# B&R Automation Studio project mappCleanUp
Automation Studio 4.10.6.39 SP

## Configuration Config1

CPU PC_any, AutomationRuntime B4.91, Build 4.1.2, Vc V4.73.0

### Task classes (Cpu.sw)
```
Cyclic#8 (cycle 10000 us):
  mappCleanU <- mappCleanUp.prg
Binaries: FWRules, TCData, udbdef, asfw, User, iomap, sysconf, arconfig, ashwd, Role, ashwac
Libraries: sys_lib, runtime, FileIO, AsBrStr, IecCheck, standard, asieccon, astime
```

### Hardware
```
PC : PC_any v1.1.1.0 (OrderNumber=PC)
  ConfigurationID = mappCleanUp_Config1
  Cyclic8Duration = 10000
  FileDevice1
  FileDeviceName1 = USER_PATH
  FileDevicePath1 = c:\Temp\CleanUpTest
```

## Configuration Simulation

CPU PC_any, AutomationRuntime M4.93, Build 4.1.2, Vc V4.73.0

### Hardware
```
PC : PC_any v1.1.1.0 (OrderNumber=PC)
  ConfigurationID = mappCleanUp_Config1
  Cyclic8Duration = 10000
  FileDevice1
  FileDeviceName1 = USER
  FileDevicePath1 = c:\Temp\CleanUpTest
```

## Configuration X20CP

CPU X20CP3687X, AutomationRuntime M4.93, Build 4.1.2, Vc V4.73.3

### Task classes (Cpu.sw)
```
Cyclic#8:
  mappCleanU <- mappCleanUp.prg
Libraries: operator, runtime, astime, AsIecCon, sys_lib, FileIO, AsBrStr, IecCheck, standard
```

### Hardware
```
X20CP3687X : X20CP3687X v1.8.2.0
  Connector IF2:
    ActivateDevice = 1
    ActivateSnmp = 2
  ConfigurationID = mappCleanUp_X20CP
  FileDevice1
  FileDeviceName1 = USER
  FileDevicePath1 = USER_PATH
  FtpUser1
  FtpUsername1 = admin
  FtpUserPassword1 = +ZKvy1J8o41WeGJ4ICTiSOGGvLAHu+nBthxiKzD2AAg=  // admin
  FtpUserSalt1 = TuKBiUW7
  FTPAccessRight1 = 0
```

## Logical view

Binary libraries used (declarations not repeated): operator, runtime, astime, AsIecCon, sys_lib, FileIO, AsBrStr, IecCheck, standard


### Program Logical/mappCleanUp (IEC)

#### Main.st - Init, cyclic, exit code
```iecst
PROGRAM _INIT
	(* Insert code here *)

END_PROGRAM

PROGRAM _CYCLIC
	CASE State OF
		CLEANUP_WAIT:
			CleanUp.Status := ERR_OK;

			DevMemInfo_0.enable := FALSE;
			DevMemInfo_0();
			DirInfo_0.enable := FALSE;
			DirInfo_0();
			DirOpen_0.enable := FALSE;
			DirOpen_0();
			DirReadEx_0.enable := FALSE;
			DirReadEx_0();
			DirClose_0.enable := FALSE;
			DirClose_0();
			FileDelete_0.enable := FALSE;
			FileDelete_0();

			// Command delete oldest file
			IF EDGEPOS(CleanUp.CMD.DeleteOldest) THEN
				// Reset variables
				brsmemset(ADR(CleanUp.DAT), 0, SIZEOF(CleanUp.DAT));
				brsmemset(ADR(FileInformation), 0, SIZEOF(FileInformation));

				// Set callbacks and status
				StateAfterInfo := CLEANUP_DIR_INFO;
				StateAfterRead := CLEANUP_DELETE_OLDEST;
				StateAfterDelete := CLEANUP_DIR_CLOSE;
				CleanUp.Status := ERR_FUB_BUSY;

				State := CLEANUP_MEM_INFO;
			END_IF

			// Command delete oldest than
			IF EDGEPOS(CleanUp.CMD.DeleteOlderThan) THEN
				IF CleanUp.PAR.OlderThan <> DT#1970-01-01-00:00:00 THEN
					// Reset variables
					brsmemset(ADR(CleanUp.DAT), 0, SIZEOF(CleanUp.DAT));
					brsmemset(ADR(FileInformation), 0, SIZEOF(FileInformation));

					// Set callbacks and status
					StateAfterInfo := CLEANUP_DIR_INFO;
					StateAfterRead := CLEANUP_DELETE_OLDER_THAN;
					StateAfterDelete := CLEANUP_DIR_READ;
					CleanUp.Status := ERR_FUB_BUSY;

					State := CLEANUP_MEM_INFO;
				ELSE
					State := CreateError(ADR(CleanUp), CLEANUP_ERR_PAR_IS_EMPTY, 'parameter >OlderThan< was not set', State, ADR(Logger));
				END_IF
			END_IF

			// Command delete files and keep x
			IF EDGEPOS(CleanUp.CMD.DeleteMaxFiles) THEN
				IF CleanUp.PAR.MaxFilesToKeep <> 0 THEN
					// Reset variables
					brsmemset(ADR(CleanUp.DAT), 0, SIZEOF(CleanUp.DAT));
					brsmemset(ADR(FileInformation), 0, SIZEOF(FileInformation));
					SimFileCount := 0;

					// Set callbacks and status
					StateAfterInfo := CLEANUP_DIR_INFO;
					StateAfterRead := CLEANUP_DELETE_MAX_FILES_1;
					StateAfterDelete := CLEANUP_DELETE_MAX_FILES_2;

					CleanUp.Status := ERR_FUB_BUSY;

					State := CLEANUP_MEM_INFO;
				ELSE
					State := CreateError(ADR(CleanUp), CLEANUP_ERR_PAR_IS_EMPTY, 'parameter >MaxFilesToKeep< was not set', State, ADR(Logger));
				END_IF
			END_IF

			// Command delete files until minimum memory is restored
			IF EDGEPOS(CleanUp.CMD.DeleteMinSpace) THEN
				IF CleanUp.PAR.MinSpace <> 0 THEN
					// Reset variables
					brsmemset(ADR(CleanUp.DAT), 0, SIZEOF(CleanUp.DAT));
					brsmemset(ADR(FileInformation), 0, SIZEOF(FileInformation));
					SimMemCount := 0;

					// Set callbacks and status
					StateAfterInfo := CLEANUP_DIR_INFO;
					StateAfterRead := CLEANUP_DELETE_MIN_SPACE_1;
					StateAfterDelete := CLEANUP_DELETE_MIN_SPACE_2;

					CleanUp.Status := ERR_FUB_BUSY;

					State := CLEANUP_MEM_INFO;
				ELSE
					State := CreateError(ADR(CleanUp), CLEANUP_ERR_PAR_IS_EMPTY, 'parameter >MinSpace< was not set', State, ADR(Logger));
				END_IF
			END_IF

			// Command update free space
			IF EDGEPOS(CleanUp.CMD.UpdateFreeSpace) THEN
				// Set callbacks
				StateAfterInfo := CLEANUP_WAIT;

				State := CLEANUP_MEM_INFO;
			END_IF

			// -------------------------------------------------------------------------------------------
			// Get device information
		CLEANUP_MEM_INFO:
			DevMemInfo_0.enable := TRUE;
			DevMemInfo_0.pDevice := ADR(CleanUp.PAR.Device);
			DevMemInfo_0();

			// Memory information successful
			IF DevMemInfo_0.status = ERR_OK THEN
				CleanUp.DAT.FreeSpace := DevMemInfo_0.freemem + (SimMemCount * CleanUp.PAR.Simulate);

				// Go to next step
				State := StateAfterInfo;

			// Error
			ELSIF DevMemInfo_0.status <> ERR_FUB_BUSY THEN
				TmpStr1 := 'ERR memory info > ';
				brsstrcat(ADR(TmpStr1), ADR(CleanUp.PAR.Device));
				State := CreateError(ADR(CleanUp), DevMemInfo_0.status, TmpStr1, State, ADR(Logger));
			END_IF

			// -------------------------------------------------------------------------------------------
			// Get folder information
		CLEANUP_DIR_INFO:
			DirInfo_0.enable := TRUE;
			DirInfo_0.pDevice := ADR(CleanUp.PAR.Device);
			DirInfo_0.pPath := ADR(CleanUp.PAR.Path);
			DirInfo_0();

			// Dir info successful
			IF DirInfo_0.status = ERR_OK THEN
				CleanUp.DAT.FilesCount := DirInfo_0.filenum;

				// Go to next step
				State := CLEANUP_DIR_OPEN;

			// Error
			ELSIF DirInfo_0.status <> ERR_FUB_BUSY THEN
				TmpStr1 := 'ERR dir info > ';
				brsstrcat(ADR(TmpStr1), ADR(CleanUp.PAR.Device));
				brsstrcat(ADR(TmpStr1), ADR(' with dir > '));
				brsstrcat(ADR(TmpStr1), ADR(CleanUp.PAR.Path));
				State := CreateError(ADR(CleanUp), DirInfo_0.status, TmpStr1, State, ADR(Logger));
			END_IF

			// -------------------------------------------------------------------------------------------
			// Start reading folder
		CLEANUP_DIR_OPEN:
			DirOpen_0.enable := TRUE;
			DirOpen_0.pDevice := ADR(CleanUp.PAR.Device);
			DirOpen_0.pName := ADR(CleanUp.PAR.Path);
			DirOpen_0();

			// Dir open successful
			IF DirOpen_0.status = ERR_OK THEN
				// Generate log entry
				TmpStr1 := 'open device > ';
				brsstrcat(ADR(TmpStr1), ADR(CleanUp.PAR.Device));
				brsstrcat(ADR(TmpStr1), ADR(' with dir > '));
				brsstrcat(ADR(TmpStr1), ADR(CleanUp.PAR.Path));
				CreateLoggerEntry(ADR(TmpStr1), ADR(Logger));

				// Go to next step
				State := CLEANUP_DIR_READ;

				// Error
			ELSIF DirOpen_0.status <> ERR_FUB_BUSY THEN
				TmpStr1 := 'ERR open device > ';
				brsstrcat(ADR(TmpStr1), ADR(CleanUp.PAR.Device));
				brsstrcat(ADR(TmpStr1), ADR(' with dir > '));
				brsstrcat(ADR(TmpStr1), ADR(CleanUp.PAR.Path));
				State := CreateError(ADR(CleanUp), DirOpen_0.status, TmpStr1, State, ADR(Logger));
			END_IF

			// -------------------------------------------------------------------------------------------
			// Start reading folder
		CLEANUP_DIR_READ:
			DirReadEx_0.enable := TRUE;
			DirReadEx_0.ident := DirOpen_0.ident;
			DirReadEx_0.pData := ADR(FileDirInfo);
			DirReadEx_0.data_len := SIZEOF(FileDirInfo);
			DirReadEx_0();

			// New file found
			IF DirReadEx_0.status = ERR_OK AND FileDirInfo.Mode = fiFILE THEN
				IF brsstrcmp(ADR(FileDirInfo.Filename), ADR('.')) <> 0 AND brsstrcmp(ADR(FileDirInfo.Filename), ADR('..')) <> 0 THEN

					// Check if file name matches pattern
					IF IsInstr(ADR(FileDirInfo.Filename), ADR(CleanUp.PAR.Pattern)) OR CleanUp.PAR.Pattern = '' THEN
						// Generate log entry
						TmpStr1 := 'found file > ';
						brsstrcat(ADR(TmpStr1), ADR(FileDirInfo.Filename));
						CreateLoggerEntry(ADR(TmpStr1), ADR(Logger));

						// Go to next state
						State := StateAfterRead;
					ELSE
						// Generate log entry
						TmpStr1 := 'file does not match pattern > ';
						brsstrcat(ADR(TmpStr1), ADR(FileDirInfo.Filename));
						CreateLoggerEntry(ADR(TmpStr1), ADR(Logger));
					END_IF

					DirReadEx_0.enable := FALSE;
					DirReadEx_0();

				END_IF

			// No more entries
			ELSIF DirReadEx_0.status = fiERR_NO_MORE_ENTRIES THEN
				// Generate log entry
				CreateLoggerEntry(ADR('no more files found '), ADR(Logger));

				// Go to next state
				State := StateAfterRead;

				// Error
			ELSIF DirReadEx_0.status <> ERR_OK AND DirReadEx_0.status <> ERR_FUB_BUSY THEN
				TmpStr1 := 'ERR open file > ';
				brsstrcat(ADR(TmpStr1), ADR(FileDirInfo.Filename));
				State := CreateError(ADR(CleanUp), DirReadEx_0.status, TmpStr1, State, ADR(Logger));
			END_IF

			// -------------------------------------------------------------------------------------------
			// Delete oldest file
		CLEANUP_DELETE_OLDEST:
			// Evaluate next file
			IF DirReadEx_0.status <> fiERR_NO_MORE_ENTRIES THEN
				// File must be older than last
				IF FileInformation.Date > FileDirInfo.Date OR FileInformation.Date = DT#1970-01-01-00:00:00 THEN
					// Pretend that files were delete in simulation mode
					IF CleanUp.PAR.Simulate AND i < SIZEOF(CleanUp.DAT.FilesList)/SIZEOF(CleanUp.DAT.FilesList[0]) THEN
						i := 0;
						WHILE i <= CleanUp.DAT.FilesDeleted DO
							IF brsstrcmp(ADR(CleanUp.DAT.FilesList[i]), ADR(FileDirInfo.Filename)) = 0 THEN
								EXIT;
							END_IF
							i := i + 1;
						END_WHILE;
					ELSE
						i := CleanUp.DAT.FilesDeleted + 1;
					END_IF
					IF i = CleanUp.DAT.FilesDeleted + 1 THEN
						FileInformation := FileDirInfo;
					END_IF
				END_IF
				State := CLEANUP_DIR_READ;

			// Delete oldest file
			ELSE
				// Make sure we found at least one entry
				IF FileInformation.Date <> DT#1970-01-01-00:00:00 THEN
					// Fake simulation values
					IF CleanUp.PAR.Simulate THEN
						SimFileCount := SimFileCount + 1;
						SimMemCount := SimMemCount + FileInformation.Filelength;
					END_IF
					brsstrcpy(ADR(FileDeleteName), ADR(FileInformation.Filename));
					State := CLEANUP_FILE_DELETE;
				ELSE
					// Create error when there are not enough files to delete
					IF CleanUp.CMD.DeleteMinSpace AND DevMemInfo_0.freemem + SimMemCount < CleanUp.PAR.MinSpace THEN
						State := CreateError(ADR(CleanUp), CLEANUP_ERR_MIN_SPACE, 'Minimum space could not be achieved', State, ADR(Logger));
					ELSIF CleanUp.CMD.DeleteMaxFiles AND DirInfo_0.filenum - SimFileCount > CleanUp.PAR.MaxFilesToKeep THEN
						State := CreateError(ADR(CleanUp), CLEANUP_ERR_MIN_FILES, 'Minimum file count could not be achieved', State, ADR(Logger));
					ELSE
						State := CLEANUP_DIR_CLOSE;
					END_IF
				END_IF
			END_IF

			// -------------------------------------------------------------------------------------------
			// Delete files older than x
		CLEANUP_DELETE_OLDER_THAN:
			// Read next file, remember oldest file
			IF DirReadEx_0.status <> fiERR_NO_MORE_ENTRIES THEN
				IF FileDirInfo.Date > CleanUp.PAR.OlderThan THEN
					brsstrcpy(ADR(FileDeleteName), ADR(FileDirInfo.Filename));
					FileInformation := FileDirInfo;
					State := CLEANUP_FILE_DELETE;
				ELSE
					State := CLEANUP_DIR_READ;
				END_IF

				// Finish deleting old files
			ELSE
				State := CLEANUP_DIR_CLOSE;
			END_IF

			// -------------------------------------------------------------------------------------------
			// Delete files and keep x
		CLEANUP_DELETE_MAX_FILES_1:
			// Read next file, remember oldest file
			IF DirInfo_0.filenum - SimFileCount > CleanUp.PAR.MaxFilesToKeep THEN
				StateAfterRead := CLEANUP_DELETE_OLDEST;
				State := CLEANUP_DELETE_OLDEST;

			// Finish deleting old files
			ELSE
				State := CLEANUP_DIR_CLOSE;
			END_IF

			// -------------------------------------------------------------------------------------------
			// Delete files and keep x
		CLEANUP_DELETE_MAX_FILES_2:
			brsmemset(ADR(FileInformation), 0, SIZEOF(FileInformation));
			DirInfo_0.enable := FALSE;
			DirInfo_0();

			StateAfterRead := CLEANUP_DELETE_MAX_FILES_1;
			State := CLEANUP_DIR_INFO;

			// -------------------------------------------------------------------------------------------
			// Delete files until minimum free space is restored
		CLEANUP_DELETE_MIN_SPACE_1:
			// Read next file, remember oldest file
			IF DevMemInfo_0.freemem + SimMemCount < CleanUp.PAR.MinSpace THEN
				StateAfterRead := CLEANUP_DELETE_OLDEST;
				State := CLEANUP_DELETE_OLDEST;

			// Finish deleting old files
			ELSE
				State := CLEANUP_DIR_CLOSE;
			END_IF

			// -------------------------------------------------------------------------------------------
			// Delete files until minimum free space is restored
		CLEANUP_DELETE_MIN_SPACE_2:
			brsmemset(ADR(FileInformation), 0, SIZEOF(FileInformation));
			DirInfo_0.enable := FALSE;
			DirInfo_0();

			StateAfterRead := CLEANUP_DELETE_MIN_SPACE_1;
			State := CLEANUP_MEM_INFO;

			// -------------------------------------------------------------------------------------------
			// Close dir read
		CLEANUP_DIR_CLOSE:
			DirClose_0.enable := TRUE;
			DirClose_0.ident := DirOpen_0.ident;
			DirClose_0();

			// Directory closed successful
			IF DirClose_0.status = ERR_OK THEN
				// Generate log entry
				TmpStr1 := 'close dir ok > ';
				brsstrcat(ADR(TmpStr1), ADR(CleanUp.PAR.Path));
				CreateLoggerEntry(ADR(TmpStr1), ADR(Logger));

				StateAfterInfo := CLEANUP_WAIT;
				State := CLEANUP_MEM_INFO;

				// Error
			ELSIF DirClose_0.status <> ERR_FUB_BUSY THEN
				TmpStr1 := 'ERR open file > ';
				brsstrcat(ADR(TmpStr1), ADR(CleanUp.PAR.Path));
				State := CreateError(ADR(CleanUp), DirClose_0.status, TmpStr1, State, ADR(Logger));
			END_IF

			// -------------------------------------------------------------------------------------------
			// Delete file
		CLEANUP_FILE_DELETE:
			// Make sure file and path fit into string
			IF brsstrlen(ADR(FileDeleteName)) + brsstrlen(ADR(CleanUp.PAR.Path)) <= FILE_NAME_LEN THEN
				// Create full file name path
				TmpStr2 := CleanUp.PAR.Path;
				brsstrcat(ADR(TmpStr2), ADR('\\'));
				brsstrcat(ADR(TmpStr2), ADR(FileDeleteName));

				// Delete file
				FileDelete_0.enable := NOT CleanUp.PAR.Simulate;
				FileDelete_0.pDevice := ADR(CleanUp.PAR.Device);
				FileDelete_0.pName := ADR(TmpStr2);
				FileDelete_0();

				// File delete successful
				IF FileDelete_0.status = ERR_OK OR CleanUp.PAR.Simulate THEN
					FileDelete_0.enable := FALSE;
					FileDelete_0();

					// Generate log entry
					IF CleanUp.PAR.Simulate THEN
						TmpStr1 := 'sim delete file ok > ';
					ELSE
						TmpStr1 := 'delete file ok > ';
					END_IF
					brsstrcat(ADR(TmpStr1), ADR(FileDeleteName));
					CreateLoggerEntry(ADR(TmpStr1), ADR(Logger));

					// Remember deleted files name and count
					IF CleanUp.DAT.FilesDeleted < SIZEOF(CleanUp.DAT.FilesList)/SIZEOF(CleanUp.DAT.FilesList[0]) THEN
						CleanUp.DAT.FilesList[CleanUp.DAT.FilesDeleted] := FileDeleteName;
					END_IF
					CleanUp.DAT.FilesDeleted := CleanUp.DAT.FilesDeleted + 1;

					State := StateAfterDelete;

					// Error
				ELSIF FileDelete_0.status <> ERR_FUB_BUSY THEN
					TmpStr1 := 'ERR delete file > ';
					brsstrcat(ADR(TmpStr1), ADR(FileDeleteName));
					State := CreateError(ADR(CleanUp), FileDelete_0.status, TmpStr1, State, ADR(Logger));
				END_IF

			// File name and path are too long
			ELSE
				TmpStr1 := 'ERR file name is too long > ';
				brsstrcat(ADR(TmpStr1), ADR(FileDeleteName));
				State := CreateError(ADR(CleanUp), CLEANUP_ERR_FILE_NAME_TO_LONG, FileDeleteName, State, ADR(Logger));
			END_IF

			// -------------------------------------------------------------------------------------------
			// Error state
		CLEANUP_ERR:
			IF CleanUp.CMD.ErrorReset THEN
				brsmemset(ADR(CleanUp.ERR), 0, SIZEOF(CleanUp.ERR));

				State := CLEANUP_WAIT;
			END_IF
	END_CASE;

END_PROGRAM

PROGRAM _EXIT
	(* Insert code here *)

END_PROGRAM
```

#### Types.typ - Local data types
```iecst
TYPE
	mappCleanUpType : 	STRUCT
		CMD : mappCleanUpCmdType;
		PAR : mappCleanUpParType;
		DAT : mappCleanUpDatType;
		ERR : mappCleanUpErrType;
		Status : UINT;
	END_STRUCT;
	mappCleanUpCmdType : 	STRUCT
		DeleteMaxFiles : BOOL;
		DeleteMinSpace : BOOL;
		DeleteOldest : BOOL;
		DeleteOlderThan : BOOL;
		UpdateFreeSpace : BOOL;
		ErrorReset : BOOL;
	END_STRUCT;
	mappCleanUpParType : 	STRUCT
		Simulate : BOOL; (*Files are only listed but not acutually deleted*)
		Device : STRING[80]; (*Device name*)
		Path : STRING[200]; (*Path to files*)
		MaxFilesToKeep : UINT; (*Maximum number of files to keep*)
		MinSpace : UDINT; (*Delete files until minimum space is available*)
		OlderThan : DATE_AND_TIME; (*Delete all files older than this date*)
		Pattern : STRING[80]; (*File must match this pattern (ex. .pdf or .csv)*)
	END_STRUCT;
	mappCleanUpDatType : 	STRUCT
		FilesList : ARRAY[0..9]OF STRING[50]; (*List of files that were deleted*)
		FilesDeleted : UINT; (*Number of files that were deleted*)
		FilesCount : UDINT; (*Number of files that were deleted*)
		FreeSpace : UDINT;
	END_STRUCT;
	mappCleanUpErrType : 	STRUCT
		State : CLEANUP_STATE;
		Text : STRING[200];
	END_STRUCT;
	CLEANUP_STATE :
		(
		CLEANUP_WAIT,
		CLEANUP_MEM_INFO,
		CLEANUP_DIR_INFO,
		CLEANUP_DIR_OPEN,
		CLEANUP_DIR_READ,
		CLEANUP_DIR_CLOSE,
		CLEANUP_DELETE_OLDEST,
		CLEANUP_DELETE_OLDER_THAN,
		CLEANUP_DELETE_MAX_FILES_1,
		CLEANUP_DELETE_MAX_FILES_2,
		CLEANUP_DELETE_MIN_SPACE_1,
		CLEANUP_DELETE_MIN_SPACE_2,
		CLEANUP_FILE_DELETE,
		CLEANUP_ERR
		);
END_TYPE
```

#### Variables.var - Local variables
```iecst
VAR
	CleanUp : mappCleanUpType := (PAR:=(Simulate:=TRUE,Device:='USER',MaxFilesToKeep:=10,MinSpace:=1000000)); (*Main structure*)
END_VAR
(*-----------------------------------------------------------------------------------------------------------------------------------------------------------------------------------------------------------------------------------------------------------------------------------------*)
(*Local variables*)
VAR
	State : CLEANUP_STATE;
	StateAfterRead : CLEANUP_STATE;
	StateAfterDelete : CLEANUP_STATE;
	StateAfterInfo : CLEANUP_STATE;
	Logger : ARRAY[0..LOG_NUM] OF STRING[LOG_LEN];
	TmpStr1 : STRING[STRING_LEN];
	TmpStr2 : STRING[STRING_LEN];
	FileDeleteName : STRING[FILE_NAME_LEN];
	FileInformation : fiDIR_READ_EX_DATA;
	FileDirInfo : fiDIR_READ_EX_DATA;
	SimFileCount : UINT;
	SimMemCount : UDINT;
	i : UINT;
END_VAR
(*-----------------------------------------------------------------------------------------------------------------------------------------------------------------------------------------------------------------------------------------------------------------------------------------*)
(*Local functions*)
VAR
	DirInfo_0 : DirInfo;
	DevMemInfo_0 : DevMemInfo;
	DirOpen_0 : DirOpen;
	DirReadEx_0 : DirReadEx;
	DirClose_0 : DirClose;
	FileDelete_0 : FileDelete;
END_VAR
(*-----------------------------------------------------------------------------------------------------------------------------------------------------------------------------------------------------------------------------------------------------------------------------------------*)
(*Local error numbers*)
VAR CONSTANT
	CLEANUP_ERR_FILE_NAME_TO_LONG : UINT := 10000; (*File name + path exceeds maximum file name length*)
	CLEANUP_ERR_PAR_IS_EMPTY : UINT := 10001; (*Corresponding parameter for command is empty*)
	CLEANUP_ERR_MIN_SPACE : UINT := 10002; (*Minimum space could not be achieved*)
	CLEANUP_ERR_MIN_FILES : UINT := 10003; (*Minimum number of files could not be achieved*)
END_VAR
(*-----------------------------------------------------------------------------------------------------------------------------------------------------------------------------------------------------------------------------------------------------------------------------------------*)
(*Local constants*)
VAR CONSTANT
	FILE_NAME_LEN : UINT := 200; (*Maximum file name length*)
	STRING_LEN : UINT := FILE_NAME_LEN+100;
	LOG_LEN : USINT := 200;
	LOG_NUM : USINT := 20;
END_VAR
```

#### LocalFunctions.fun - Local function definition
```iecst
FUNCTION CreateError : CLEANUP_STATE
	VAR_INPUT
		CleanUp : REFERENCE TO mappCleanUpType;
		No : UINT;
		Text : STRING[200];
		State : CLEANUP_STATE;
		Logger : UDINT;
	END_VAR
END_FUNCTION

FUNCTION IsInstr : BOOL
	VAR_INPUT
		string1 : UDINT;
		string2 : UDINT;
	END_VAR
	VAR
		idx : UDINT;
	END_VAR
END_FUNCTION

FUNCTION CreateLoggerEntry : USINT
	VAR_INPUT
		LogMsg : UDINT; (*Log message*)
		LogBuffer : UDINT; (*Address of log buffer*)
	END_VAR
	VAR
		RtcGettime : RTCtime_typ;
		TmpStr : STRING[20];
		LastMsg : STRING[STRING_LEN];
	END_VAR
END_FUNCTION
```

#### LocalFunctions.st - Local function code
```iecst
// -------------------------------------------------------------------------------------------
// Create error
// -------------------------------------------------------------------------------------------
FUNCTION CreateError
	CleanUp.Status := No;
	CleanUp.ERR.State := State;
	CleanUp.ERR.Text := Text;

	CreateLoggerEntry(ADR(Text), Logger);

	CreateError := CLEANUP_ERR;
END_FUNCTION

// -------------------------------------------------------------------------------------------
// Is second string in first string
// -------------------------------------------------------------------------------------------
FUNCTION IsInstr
	IF (brsstrlen(string1) > brsstrlen(string2)) THEN
		FOR idx:=0 TO brsstrlen(string1) - brsstrlen(string2) DO
			IF (brsmemcmp(string1 + idx, string2, brsstrlen(string2)) = 0) THEN
				IsInstr := TRUE;
				EXIT;
			END_IF
		END_FOR;
	END_IF
END_FUNCTION

// -------------------------------------------------------------------------------------------
// Handle log buffer
// -------------------------------------------------------------------------------------------
FUNCTION CreateLoggerEntry
	IF LogBuffer = 0 THEN
		RETURN;
	END_IF
	// Make sure log message fits
	IF brsstrlen(LogMsg) > LOG_LEN - 20 THEN
		brsstrcpy(LogMsg, ADR('*** log meassage exceeds maximum length ***'));
		RETURN;
	END_IF
	// Check previous message
	IF brsstrlen(LogBuffer) > 19 THEN
		brsstrcpy(ADR(LastMsg), LogBuffer + 19);
	END_IF

	// Make sure we dont flood Logger
	IF brsstrcmp(LogMsg, ADR(LastMsg)) <> 0 AND LogBuffer <> 0 THEN
		// Move ring buffer around
		brsmemmove(LogBuffer+LOG_LEN+1, LogBuffer, LOG_LEN*(LOG_NUM-1));
		brsstrcpy(LogBuffer, ADR(''));
		// Create time information
		RTC_gettime(ADR(RtcGettime));
		IF(RtcGettime.day < 10) THEN
			brsstrcat(LogBuffer, ADR('0'));
		END_IF
		brsitoa(RtcGettime.day, ADR(TmpStr));
		brsstrcat(LogBuffer, ADR(TmpStr));
		brsitoa(RtcGettime.day, ADR(TmpStr));
		brsstrcat(LogBuffer, ADR('.'));
		IF(RtcGettime.month < 10) THEN
			brsstrcat(LogBuffer, ADR('0'));
		END_IF
		brsitoa(RtcGettime.month, ADR(TmpStr));
		brsstrcat(LogBuffer, ADR(TmpStr));
		brsstrcat(LogBuffer, ADR(' '));
		IF(RtcGettime.hour < 10) THEN
			brsstrcat(LogBuffer, ADR('0'));
		END_IF
		brsitoa(RtcGettime.hour, ADR(TmpStr));
		brsstrcat(LogBuffer, ADR(TmpStr));
		brsstrcat(LogBuffer, ADR(':'));
		IF(RtcGettime.minute < 10) THEN
			brsstrcat(LogBuffer, ADR('0'));
		END_IF
		brsitoa(RtcGettime.minute, ADR(TmpStr));
		brsstrcat(LogBuffer, ADR(TmpStr));
		brsstrcat(LogBuffer, ADR(':'));
		IF(RtcGettime.second < 10) THEN
			brsstrcat(LogBuffer, ADR('0'));
		END_IF
		brsitoa(RtcGettime.second, ADR(TmpStr));
		brsstrcat(LogBuffer, ADR(TmpStr));
		brsstrcat(LogBuffer, ADR('.'));
		IF(RtcGettime.millisec < 10) THEN
			brsstrcat(LogBuffer, ADR('00'));
		ELSIF(RtcGettime.millisec < 100) THEN
			brsstrcat(LogBuffer, ADR('0'));
		END_IF
		brsitoa(RtcGettime.millisec, ADR(TmpStr));
		brsstrcat(LogBuffer, ADR(TmpStr));
		// Add log message
		brsstrcat(LogBuffer, ADR(' '));
		brsstrcat(LogBuffer, LogMsg);
	END_IF

	CreateLoggerEntry := TRUE;
END_FUNCTION
```

#### revision.txt
```
Version 0.1

First public release
```

Listed in the project but not available here: Logical/Global.typ, Logical/Global.var
